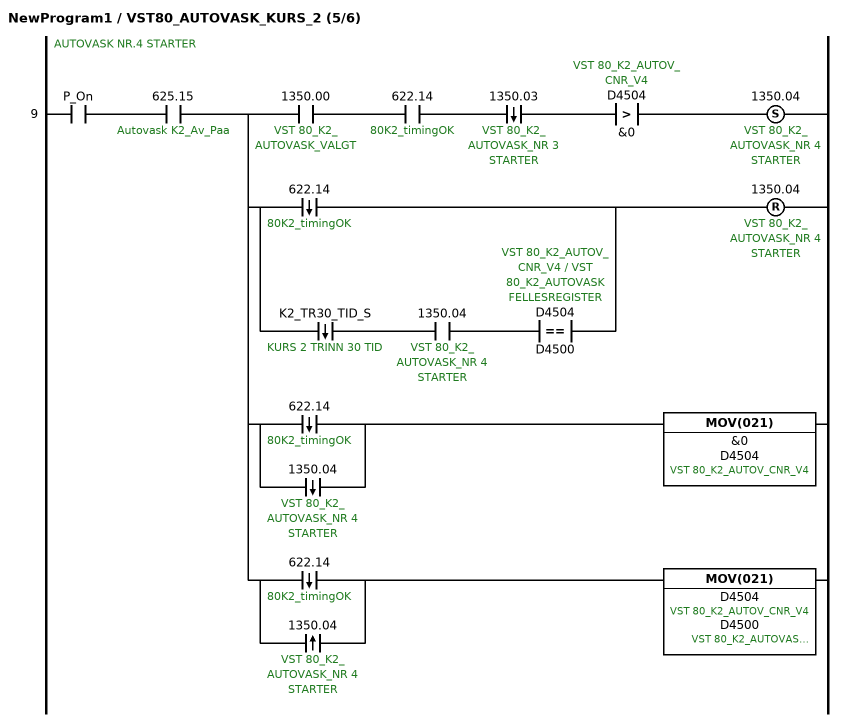
; [picture p288: NewProgram1 / VST80_AUTOVASK_KURS_2, rungs 9-9]
; rung 9: AUTOVASK NR.4 STARTER
LD P_On
AND 625.15  ; Autovask K2_Av_Paa
OUT TR0
AND 1350.00  ; VST 80_K2_AUTOVASK_VALGT
AND 622.14  ; 80K2_timingOK
%AND 1350.03  ; VST 80_K2_AUTOVASK_NR 3 STARTER
AND>(320) D4504 &0  ; VST 80_K2_AUTOV_CNR_V4
SET 1350.04  ; VST 80_K2_AUTOVASK_NR 4 STARTER
LD TR0
%LD 622.14  ; 80K2_timingOK
%LD K2_TR30_TID_S  ; KURS 2 TRINN 30 TID
AND 1350.04  ; VST 80_K2_AUTOVASK_NR 4 STARTER
AND=(300) D4504 D4500  ; VST 80_K2_AUTOV_CNR_V4, VST 80_K2_AUTOVASK FELLESREGISTER
ORLD
ANDLD
RSET 1350.04  ; VST 80_K2_AUTOVASK_NR 4 STARTER
LD TR0
%LD 622.14  ; 80K2_timingOK
%OR 1350.04  ; VST 80_K2_AUTOVASK_NR 4 STARTER
ANDLD
MOV(021) &0 D4504  ; VST 80_K2_AUTOV_CNR_V4
LD TR0
%LD 622.14  ; 80K2_timingOK
@OR 1350.04  ; VST 80_K2_AUTOVASK_NR 4 STARTER
ANDLD
MOV(021) D4504 D4500  ; VST 80_K2_AUTOV_CNR_V4, VST 80_K2_AUTOVASK FELLESREGISTER

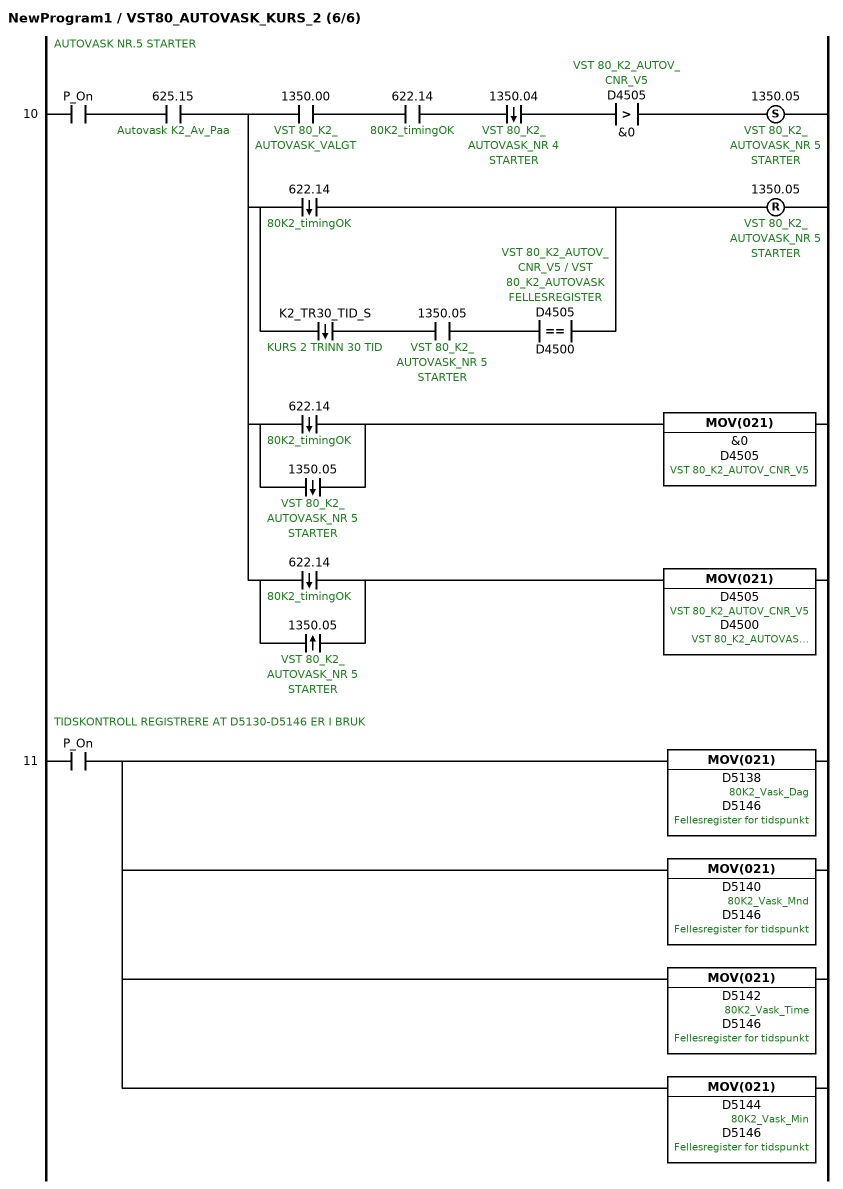
; rung 10: AUTOVASK NR.5 STARTER
LD P_On
AND 625.15  ; Autovask K2_Av_Paa
OUT TR0
AND 1350.00  ; VST 80_K2_AUTOVASK_VALGT
AND 622.14  ; 80K2_timingOK
%AND 1350.04  ; VST 80_K2_AUTOVASK_NR 4 STARTER
AND>(320) D4505 &0  ; VST 80_K2_AUTOV_CNR_V5
SET 1350.05  ; VST 80_K2_AUTOVASK_NR 5 STARTER
LD TR0
%LD 622.14  ; 80K2_timingOK
%LD K2_TR30_TID_S  ; KURS 2 TRINN 30 TID
AND 1350.05  ; VST 80_K2_AUTOVASK_NR 5 STARTER
AND=(300) D4505 D4500  ; VST 80_K2_AUTOV_CNR_V5, VST 80_K2_AUTOVASK FELLESREGISTER
ORLD
ANDLD
RSET 1350.05  ; VST 80_K2_AUTOVASK_NR 5 STARTER
LD TR0
%LD 622.14  ; 80K2_timingOK
%OR 1350.05  ; VST 80_K2_AUTOVASK_NR 5 STARTER
ANDLD
MOV(021) &0 D4505  ; VST 80_K2_AUTOV_CNR_V5
LD TR0
%LD 622.14  ; 80K2_timingOK
@OR 1350.05  ; VST 80_K2_AUTOVASK_NR 5 STARTER
ANDLD
MOV(021) D4505 D4500  ; VST 80_K2_AUTOV_CNR_V5, VST 80_K2_AUTOVASK FELLESREGISTER
; rung 11: TIDSKONTROLL REGISTRERE AT D5130-D5146 ER I BRUK
LD P_On
MOV(021) D5138 D5146  ; 80K2_Vask_Dag, Fellesregister for tidspunkt
MOV(021) D5140 D5146  ; 80K2_Vask_Mnd, Fellesregister for tidspunkt
MOV(021) D5142 D5146  ; 80K2_Vask_Time, Fellesregister for tidspunkt
MOV(021) D5144 D5146  ; 80K2_Vask_Min, Fellesregister for tidspunkt
; rung 12: Ingen_kommentar_funnet

### Section VST80_K_3_TIDER_TR1_18

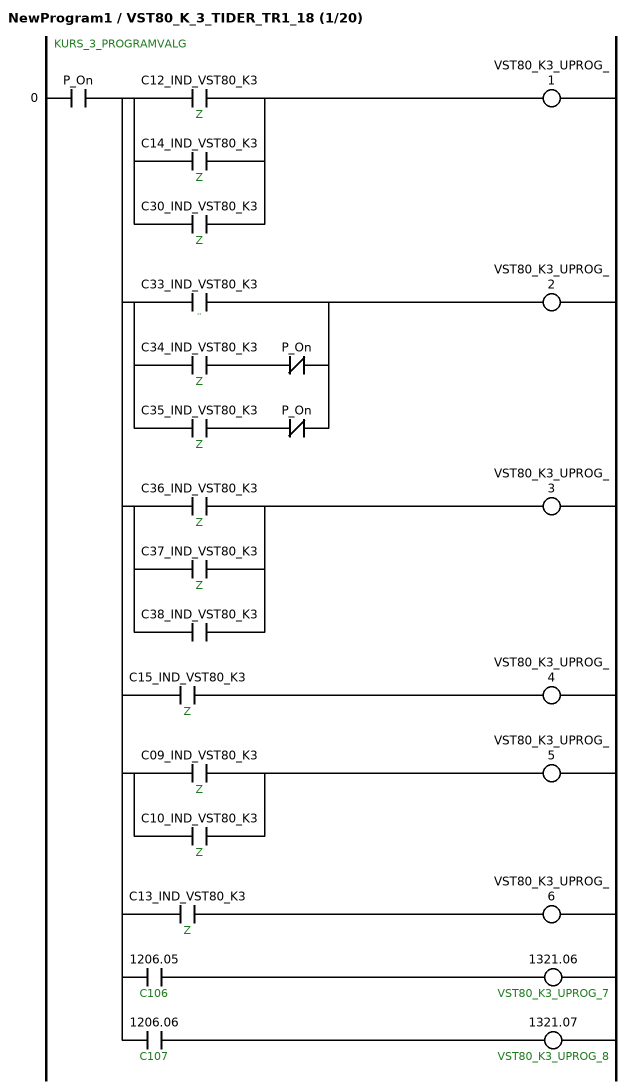
; rung 0: KURS_3_PROGRAMVALG
LD P_On
OUT TR0
LD C12_IND_VST80_K3  ; Z
OR C14_IND_VST80_K3  ; Z
OR C30_IND_VST80_K3  ; Z
ANDLD
OUT VST80_K3_UPROG_1
LD TR0
LD C33_IND_VST80_K3  ; ¨
LD C34_IND_VST80_K3  ; Z
ANDNOT P_On
ORLD
LD C35_IND_VST80_K3  ; Z
ANDNOT P_On
ORLD
ANDLD
OUT VST80_K3_UPROG_2
LD TR0
LD C36_IND_VST80_K3  ; Z
OR C37_IND_VST80_K3  ; Z
OR C38_IND_VST80_K3
ANDLD
OUT VST80_K3_UPROG_3
LD TR0
AND C15_IND_VST80_K3  ; Z
OUT VST80_K3_UPROG_4
LD TR0
LD C09_IND_VST80_K3  ; Z
OR C10_IND_VST80_K3  ; Z
ANDLD
OUT VST80_K3_UPROG_5
LD TR0
AND C13_IND_VST80_K3  ; Z
OUT VST80_K3_UPROG_6
LD TR0
AND 1206.05  ; C106
OUT 1321.06  ; VST80_K3_UPROG_7
LD TR0
AND 1206.06  ; C107
OUT 1321.07  ; VST80_K3_UPROG_8

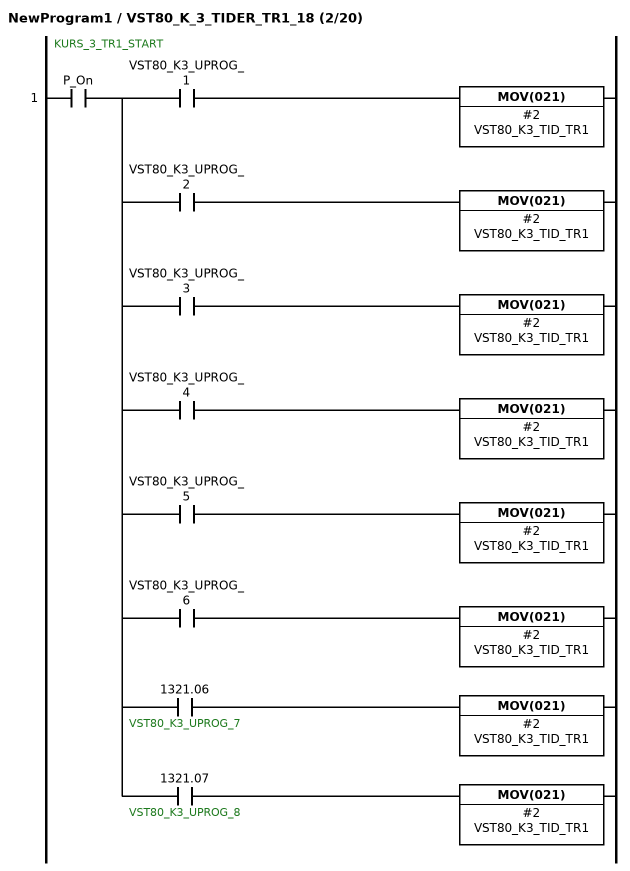
; rung 1: KURS_3_TR1_START
LD P_On
OUT TR0
AND VST80_K3_UPROG_1
MOV(021) #2 VST80_K3_TID_TR1
LD TR0
AND VST80_K3_UPROG_2
MOV(021) #2 VST80_K3_TID_TR1
LD TR0
AND VST80_K3_UPROG_3
MOV(021) #2 VST80_K3_TID_TR1
LD TR0
AND VST80_K3_UPROG_4
MOV(021) #2 VST80_K3_TID_TR1
LD TR0
AND VST80_K3_UPROG_5
MOV(021) #2 VST80_K3_TID_TR1
LD TR0
AND VST80_K3_UPROG_6
MOV(021) #2 VST80_K3_TID_TR1
LD TR0
AND 1321.06  ; VST80_K3_UPROG_7
MOV(021) #2 VST80_K3_TID_TR1
LD TR0
AND 1321.07  ; VST80_K3_UPROG_8
MOV(021) #2 VST80_K3_TID_TR1

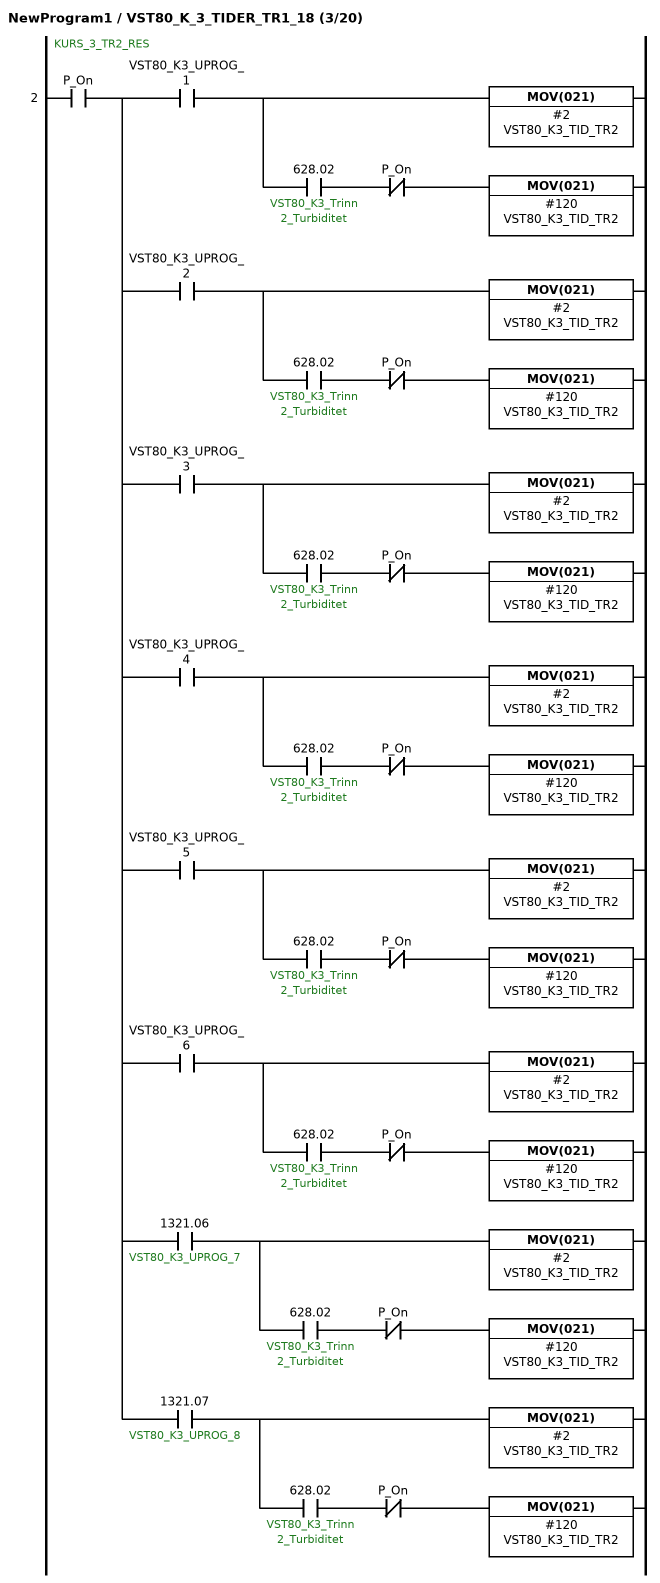
; rung 2: KURS_3_TR2_RES
LD P_On
OUT TR0
AND VST80_K3_UPROG_1
MOV(021) #2 VST80_K3_TID_TR2
AND 628.02  ; VST80_K3_Trinn 2_Turbiditet
ANDNOT P_On
MOV(021) #120 VST80_K3_TID_TR2
LD TR0
AND VST80_K3_UPROG_2
MOV(021) #2 VST80_K3_TID_TR2
AND 628.02  ; VST80_K3_Trinn 2_Turbiditet
ANDNOT P_On
MOV(021) #120 VST80_K3_TID_TR2
LD TR0
AND VST80_K3_UPROG_3
MOV(021) #2 VST80_K3_TID_TR2
AND 628.02  ; VST80_K3_Trinn 2_Turbiditet
ANDNOT P_On
MOV(021) #120 VST80_K3_TID_TR2
LD TR0
AND VST80_K3_UPROG_4
MOV(021) #2 VST80_K3_TID_TR2
AND 628.02  ; VST80_K3_Trinn 2_Turbiditet
ANDNOT P_On
MOV(021) #120 VST80_K3_TID_TR2
LD TR0
AND VST80_K3_UPROG_5
MOV(021) #2 VST80_K3_TID_TR2
AND 628.02  ; VST80_K3_Trinn 2_Turbiditet
ANDNOT P_On
MOV(021) #120 VST80_K3_TID_TR2
LD TR0
AND VST80_K3_UPROG_6
MOV(021) #2 VST80_K3_TID_TR2
AND 628.02  ; VST80_K3_Trinn 2_Turbiditet
ANDNOT P_On
MOV(021) #120 VST80_K3_TID_TR2
LD TR0
AND 1321.06  ; VST80_K3_UPROG_7
MOV(021) #2 VST80_K3_TID_TR2
AND 628.02  ; VST80_K3_Trinn 2_Turbiditet
ANDNOT P_On
MOV(021) #120 VST80_K3_TID_TR2
LD TR0
AND 1321.07  ; VST80_K3_UPROG_8
MOV(021) #2 VST80_K3_TID_TR2
AND 628.02  ; VST80_K3_Trinn 2_Turbiditet
ANDNOT P_On
MOV(021) #120 VST80_K3_TID_TR2

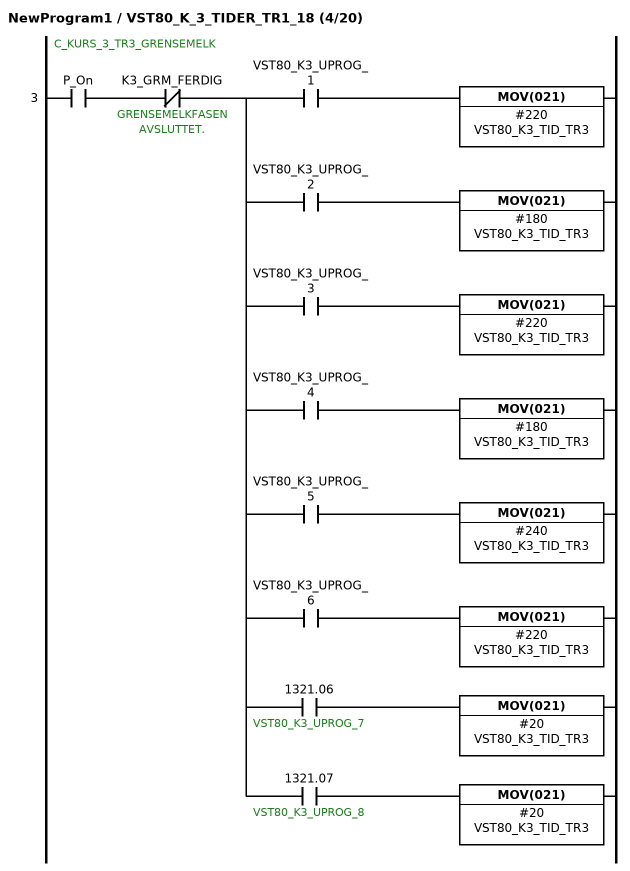
; rung 3: C_KURS_3_TR3_GRENSEMELK
LD P_On
ANDNOT K3_GRM_FERDIG  ; GRENSEMELKFASEN AVSLUTTET.
OUT TR0
AND VST80_K3_UPROG_1
MOV(021) #220 VST80_K3_TID_TR3
LD TR0
AND VST80_K3_UPROG_2
MOV(021) #180 VST80_K3_TID_TR3
LD TR0
AND VST80_K3_UPROG_3
MOV(021) #220 VST80_K3_TID_TR3
LD TR0
AND VST80_K3_UPROG_4
MOV(021) #180 VST80_K3_TID_TR3
LD TR0
AND VST80_K3_UPROG_5
MOV(021) #240 VST80_K3_TID_TR3
LD TR0
AND VST80_K3_UPROG_6
MOV(021) #220 VST80_K3_TID_TR3
LD TR0
AND 1321.06  ; VST80_K3_UPROG_7
MOV(021) #20 VST80_K3_TID_TR3
LD TR0
AND 1321.07  ; VST80_K3_UPROG_8
MOV(021) #20 VST80_K3_TID_TR3

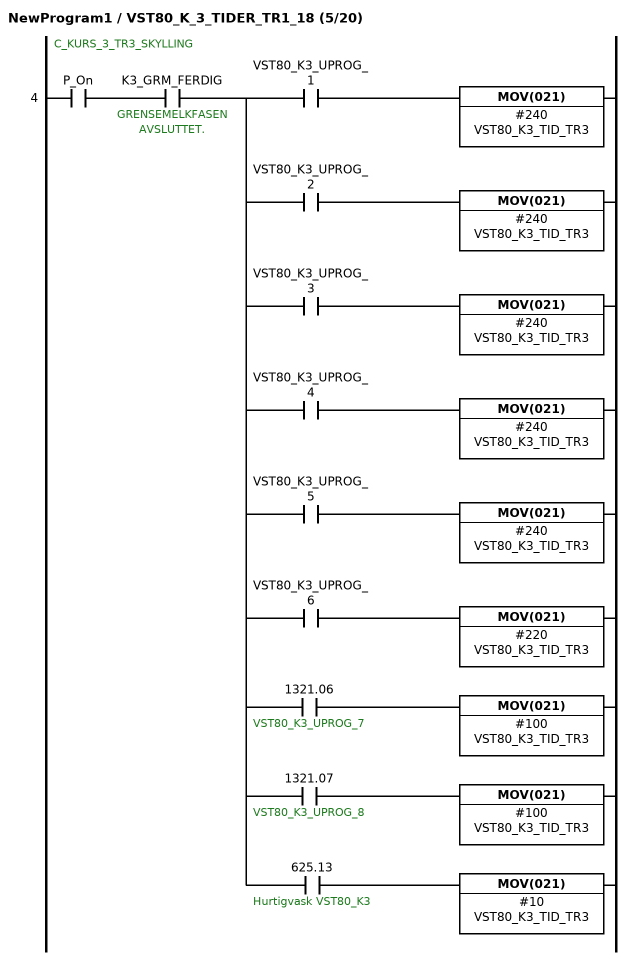
; rung 4: C_KURS_3_TR3_SKYLLING
LD P_On
AND K3_GRM_FERDIG  ; GRENSEMELKFASEN AVSLUTTET.
OUT TR0
AND VST80_K3_UPROG_1
MOV(021) #240 VST80_K3_TID_TR3
LD TR0
AND VST80_K3_UPROG_2
MOV(021) #240 VST80_K3_TID_TR3
LD TR0
AND VST80_K3_UPROG_3
MOV(021) #240 VST80_K3_TID_TR3
LD TR0
AND VST80_K3_UPROG_4
MOV(021) #240 VST80_K3_TID_TR3
LD TR0
AND VST80_K3_UPROG_5
MOV(021) #240 VST80_K3_TID_TR3
LD TR0
AND VST80_K3_UPROG_6
MOV(021) #220 VST80_K3_TID_TR3
LD TR0
AND 1321.06  ; VST80_K3_UPROG_7
MOV(021) #100 VST80_K3_TID_TR3
LD TR0
AND 1321.07  ; VST80_K3_UPROG_8
MOV(021) #100 VST80_K3_TID_TR3
LD TR0
AND 625.13  ; Hurtigvask VST80_K3
MOV(021) #10 VST80_K3_TID_TR3

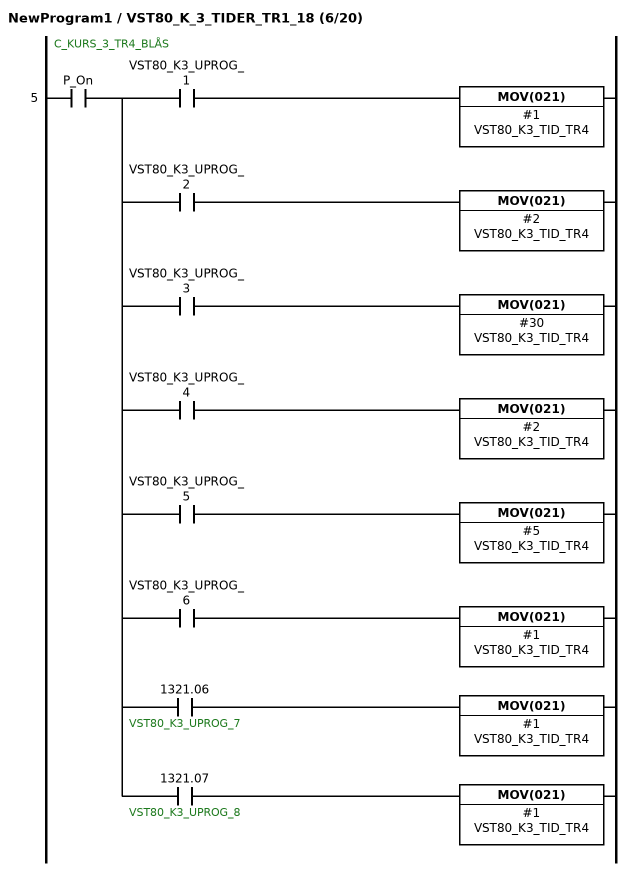
; rung 5: C_KURS_3_TR4_BLÅS
LD P_On
OUT TR0
AND VST80_K3_UPROG_1
MOV(021) #1 VST80_K3_TID_TR4
LD TR0
AND VST80_K3_UPROG_2
MOV(021) #2 VST80_K3_TID_TR4
LD TR0
AND VST80_K3_UPROG_3
MOV(021) #30 VST80_K3_TID_TR4
LD TR0
AND VST80_K3_UPROG_4
MOV(021) #2 VST80_K3_TID_TR4
LD TR0
AND VST80_K3_UPROG_5
MOV(021) #5 VST80_K3_TID_TR4
LD TR0
AND VST80_K3_UPROG_6
MOV(021) #1 VST80_K3_TID_TR4
LD TR0
AND 1321.06  ; VST80_K3_UPROG_7
MOV(021) #1 VST80_K3_TID_TR4
LD TR0
AND 1321.07  ; VST80_K3_UPROG_8
MOV(021) #1 VST80_K3_TID_TR4

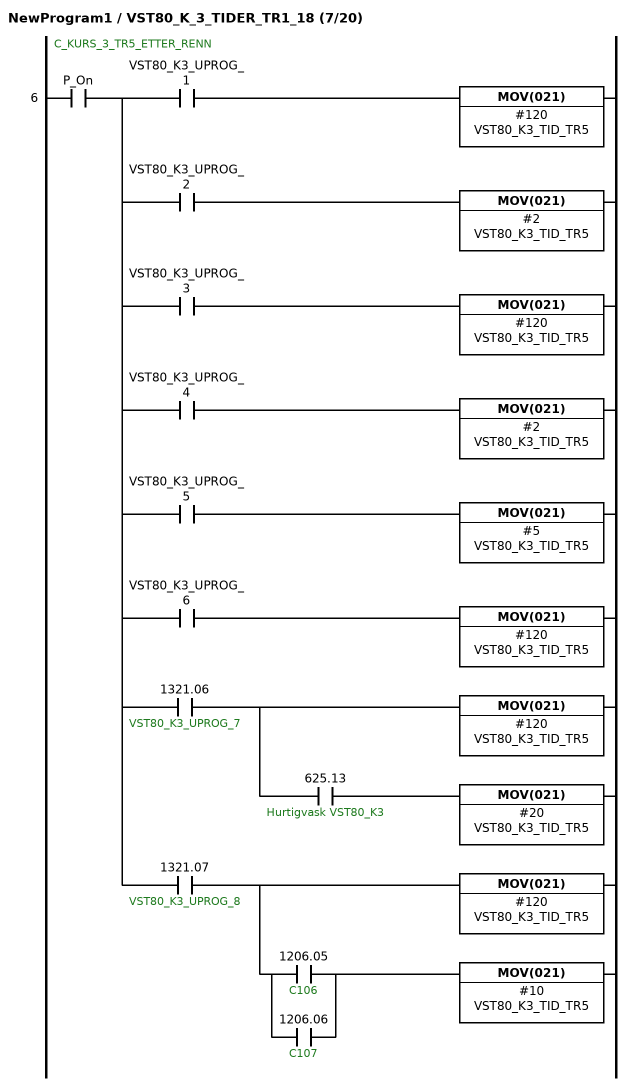
; rung 6: C_KURS_3_TR5_ETTER_RENN
LD P_On
OUT TR0
AND VST80_K3_UPROG_1
MOV(021) #120 VST80_K3_TID_TR5
LD TR0
AND VST80_K3_UPROG_2
MOV(021) #2 VST80_K3_TID_TR5
LD TR0
AND VST80_K3_UPROG_3
MOV(021) #120 VST80_K3_TID_TR5
LD TR0
AND VST80_K3_UPROG_4
MOV(021) #2 VST80_K3_TID_TR5
LD TR0
AND VST80_K3_UPROG_5
MOV(021) #5 VST80_K3_TID_TR5
LD TR0
AND VST80_K3_UPROG_6
MOV(021) #120 VST80_K3_TID_TR5
LD TR0
AND 1321.06  ; VST80_K3_UPROG_7
MOV(021) #120 VST80_K3_TID_TR5
AND 625.13  ; Hurtigvask VST80_K3
MOV(021) #20 VST80_K3_TID_TR5
LD TR0
AND 1321.07  ; VST80_K3_UPROG_8
MOV(021) #120 VST80_K3_TID_TR5
LD 1206.05  ; C106
OR 1206.06  ; C107
ANDLD
MOV(021) #10 VST80_K3_TID_TR5

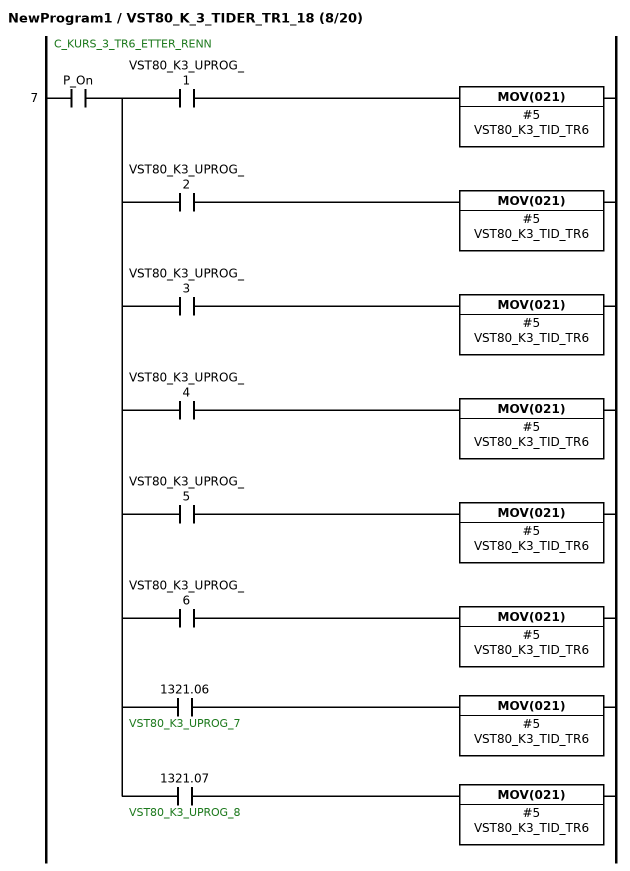
; rung 7: C_KURS_3_TR6_ETTER_RENN
LD P_On
OUT TR0
AND VST80_K3_UPROG_1
MOV(021) #5 VST80_K3_TID_TR6
LD TR0
AND VST80_K3_UPROG_2
MOV(021) #5 VST80_K3_TID_TR6
LD TR0
AND VST80_K3_UPROG_3
MOV(021) #5 VST80_K3_TID_TR6
LD TR0
AND VST80_K3_UPROG_4
MOV(021) #5 VST80_K3_TID_TR6
LD TR0
AND VST80_K3_UPROG_5
MOV(021) #5 VST80_K3_TID_TR6
LD TR0
AND VST80_K3_UPROG_6
MOV(021) #5 VST80_K3_TID_TR6
LD TR0
AND 1321.06  ; VST80_K3_UPROG_7
MOV(021) #5 VST80_K3_TID_TR6
LD TR0
AND 1321.07  ; VST80_K3_UPROG_8
MOV(021) #5 VST80_K3_TID_TR6

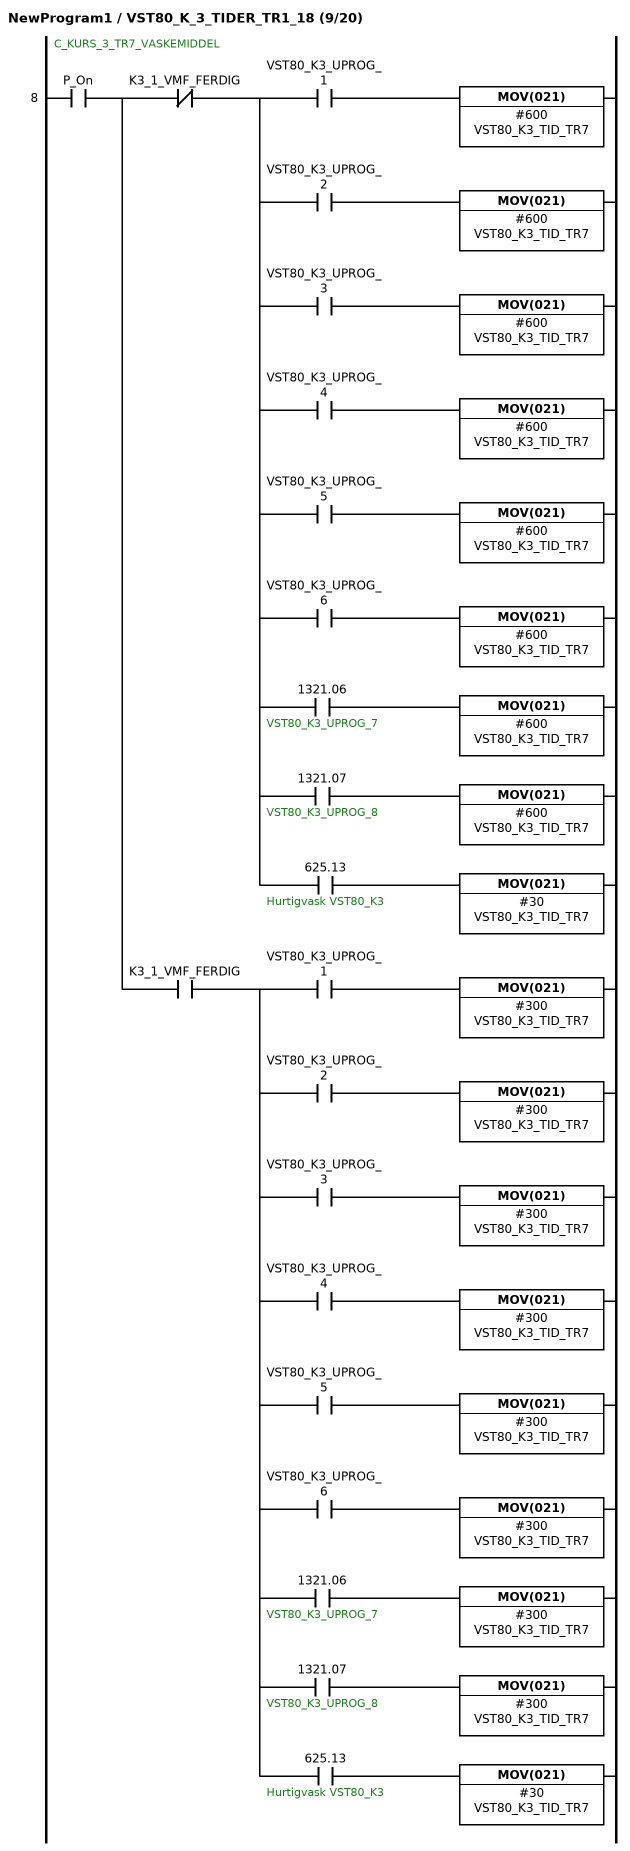
; rung 8: C_KURS_3_TR7_VASKEMIDDEL
LD P_On
OUT TR0
ANDNOT K3_1_VMF_FERDIG
OUT TR1
AND VST80_K3_UPROG_1
MOV(021) #600 VST80_K3_TID_TR7
LD TR1
AND VST80_K3_UPROG_2
MOV(021) #600 VST80_K3_TID_TR7
LD TR1
AND VST80_K3_UPROG_3
MOV(021) #600 VST80_K3_TID_TR7
LD TR1
AND VST80_K3_UPROG_4
MOV(021) #600 VST80_K3_TID_TR7
LD TR1
AND VST80_K3_UPROG_5
MOV(021) #600 VST80_K3_TID_TR7
LD TR1
AND VST80_K3_UPROG_6
MOV(021) #600 VST80_K3_TID_TR7
LD TR1
AND 1321.06  ; VST80_K3_UPROG_7
MOV(021) #600 VST80_K3_TID_TR7
LD TR1
AND 1321.07  ; VST80_K3_UPROG_8
MOV(021) #600 VST80_K3_TID_TR7
LD TR1
AND 625.13  ; Hurtigvask VST80_K3
MOV(021) #30 VST80_K3_TID_TR7
LD TR0
AND K3_1_VMF_FERDIG
OUT TR0
AND VST80_K3_UPROG_1
MOV(021) #300 VST80_K3_TID_TR7
LD TR0
AND VST80_K3_UPROG_2
MOV(021) #300 VST80_K3_TID_TR7
LD TR0
AND VST80_K3_UPROG_3
MOV(021) #300 VST80_K3_TID_TR7
LD TR0
AND VST80_K3_UPROG_4
MOV(021) #300 VST80_K3_TID_TR7
LD TR0
AND VST80_K3_UPROG_5
MOV(021) #300 VST80_K3_TID_TR7
LD TR0
AND VST80_K3_UPROG_6
MOV(021) #300 VST80_K3_TID_TR7
LD TR0
AND 1321.06  ; VST80_K3_UPROG_7
MOV(021) #300 VST80_K3_TID_TR7
LD TR0
AND 1321.07  ; VST80_K3_UPROG_8
MOV(021) #300 VST80_K3_TID_TR7
LD TR0
AND 625.13  ; Hurtigvask VST80_K3
MOV(021) #30 VST80_K3_TID_TR7

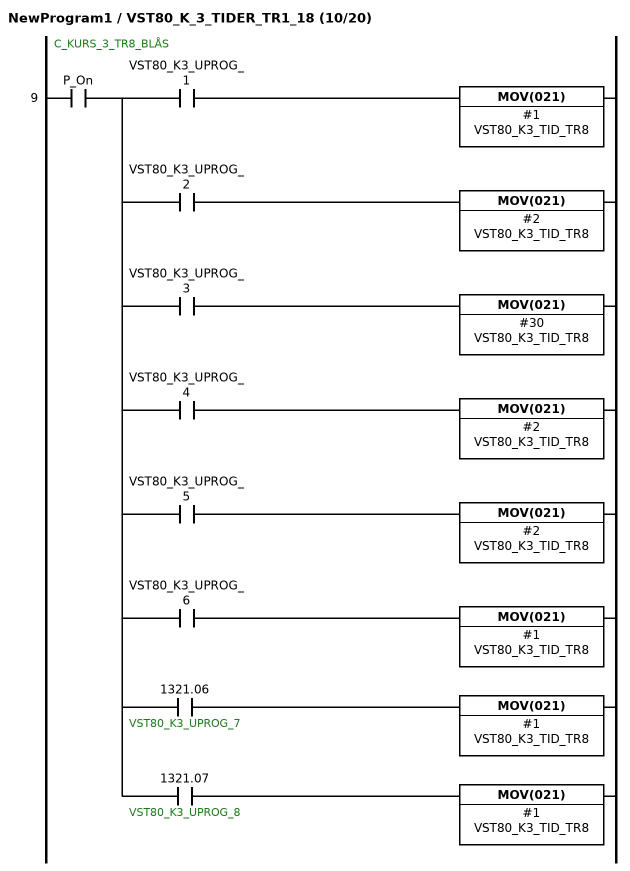
; rung 9: C_KURS_3_TR8_BLÅS
LD P_On
OUT TR0
AND VST80_K3_UPROG_1
MOV(021) #1 VST80_K3_TID_TR8
LD TR0
AND VST80_K3_UPROG_2
MOV(021) #2 VST80_K3_TID_TR8
LD TR0
AND VST80_K3_UPROG_3
MOV(021) #30 VST80_K3_TID_TR8
LD TR0
AND VST80_K3_UPROG_4
MOV(021) #2 VST80_K3_TID_TR8
LD TR0
AND VST80_K3_UPROG_5
MOV(021) #2 VST80_K3_TID_TR8
LD TR0
AND VST80_K3_UPROG_6
MOV(021) #1 VST80_K3_TID_TR8
LD TR0
AND 1321.06  ; VST80_K3_UPROG_7
MOV(021) #1 VST80_K3_TID_TR8
LD TR0
AND 1321.07  ; VST80_K3_UPROG_8
MOV(021) #1 VST80_K3_TID_TR8

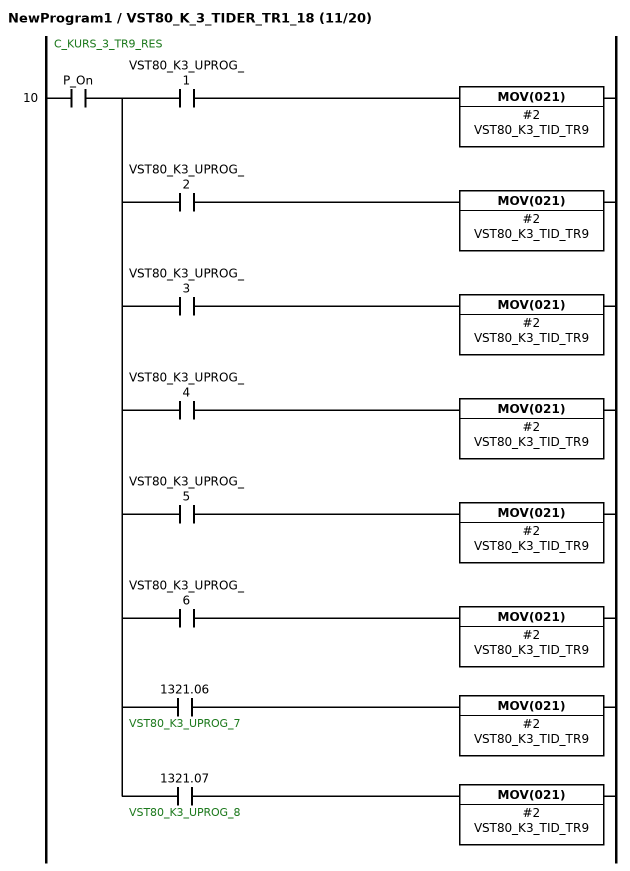
; rung 10: C_KURS_3_TR9_RES
LD P_On
OUT TR0
AND VST80_K3_UPROG_1
MOV(021) #2 VST80_K3_TID_TR9
LD TR0
AND VST80_K3_UPROG_2
MOV(021) #2 VST80_K3_TID_TR9
LD TR0
AND VST80_K3_UPROG_3
MOV(021) #2 VST80_K3_TID_TR9
LD TR0
AND VST80_K3_UPROG_4
MOV(021) #2 VST80_K3_TID_TR9
LD TR0
AND VST80_K3_UPROG_5
MOV(021) #2 VST80_K3_TID_TR9
LD TR0
AND VST80_K3_UPROG_6
MOV(021) #2 VST80_K3_TID_TR9
LD TR0
AND 1321.06  ; VST80_K3_UPROG_7
MOV(021) #2 VST80_K3_TID_TR9
LD TR0
AND 1321.07  ; VST80_K3_UPROG_8
MOV(021) #2 VST80_K3_TID_TR9

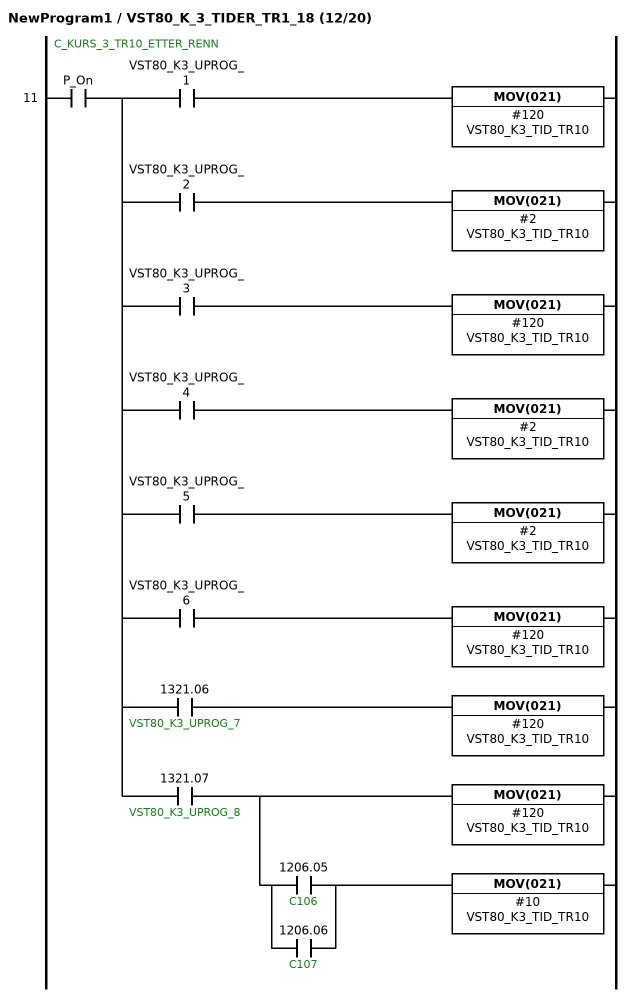
; rung 11: C_KURS_3_TR10_ETTER_RENN
LD P_On
OUT TR0
AND VST80_K3_UPROG_1
MOV(021) #120 VST80_K3_TID_TR10
LD TR0
AND VST80_K3_UPROG_2
MOV(021) #2 VST80_K3_TID_TR10
LD TR0
AND VST80_K3_UPROG_3
MOV(021) #120 VST80_K3_TID_TR10
LD TR0
AND VST80_K3_UPROG_4
MOV(021) #2 VST80_K3_TID_TR10
LD TR0
AND VST80_K3_UPROG_5
MOV(021) #2 VST80_K3_TID_TR10
LD TR0
AND VST80_K3_UPROG_6
MOV(021) #120 VST80_K3_TID_TR10
LD TR0
AND 1321.06  ; VST80_K3_UPROG_7
MOV(021) #120 VST80_K3_TID_TR10
LD TR0
AND 1321.07  ; VST80_K3_UPROG_8
MOV(021) #120 VST80_K3_TID_TR10
LD 1206.05  ; C106
OR 1206.06  ; C107
ANDLD
MOV(021) #10 VST80_K3_TID_TR10

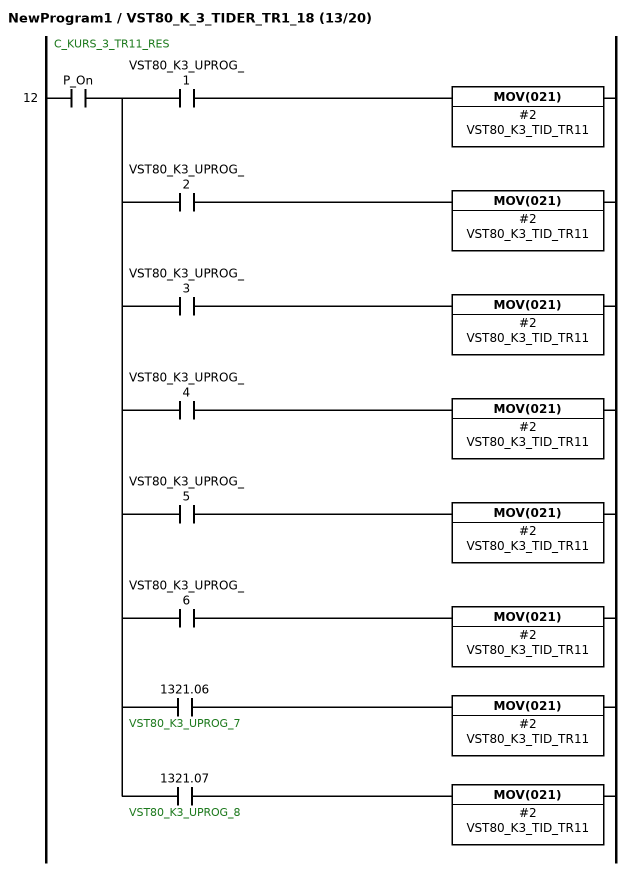
; rung 12: C_KURS_3_TR11_RES
LD P_On
OUT TR0
AND VST80_K3_UPROG_1
MOV(021) #2 VST80_K3_TID_TR11
LD TR0
AND VST80_K3_UPROG_2
MOV(021) #2 VST80_K3_TID_TR11
LD TR0
AND VST80_K3_UPROG_3
MOV(021) #2 VST80_K3_TID_TR11
LD TR0
AND VST80_K3_UPROG_4
MOV(021) #2 VST80_K3_TID_TR11
LD TR0
AND VST80_K3_UPROG_5
MOV(021) #2 VST80_K3_TID_TR11
LD TR0
AND VST80_K3_UPROG_6
MOV(021) #2 VST80_K3_TID_TR11
LD TR0
AND 1321.06  ; VST80_K3_UPROG_7
MOV(021) #2 VST80_K3_TID_TR11
LD TR0
AND 1321.07  ; VST80_K3_UPROG_8
MOV(021) #2 VST80_K3_TID_TR11

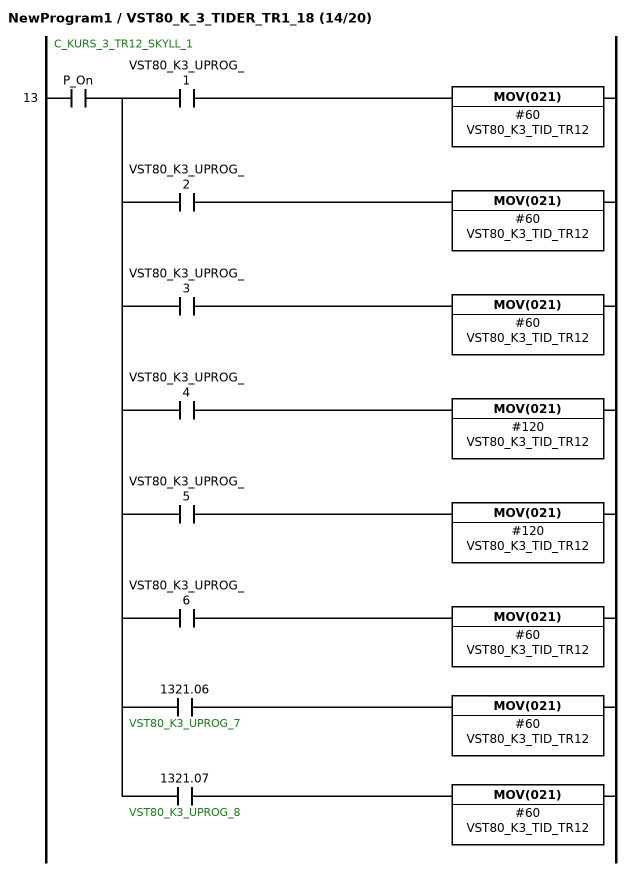
; rung 13: C_KURS_3_TR12_SKYLL_1
LD P_On
OUT TR0
AND VST80_K3_UPROG_1
MOV(021) #60 VST80_K3_TID_TR12
LD TR0
AND VST80_K3_UPROG_2
MOV(021) #60 VST80_K3_TID_TR12
LD TR0
AND VST80_K3_UPROG_3
MOV(021) #60 VST80_K3_TID_TR12
LD TR0
AND VST80_K3_UPROG_4
MOV(021) #120 VST80_K3_TID_TR12
LD TR0
AND VST80_K3_UPROG_5
MOV(021) #120 VST80_K3_TID_TR12
LD TR0
AND VST80_K3_UPROG_6
MOV(021) #60 VST80_K3_TID_TR12
LD TR0
AND 1321.06  ; VST80_K3_UPROG_7
MOV(021) #60 VST80_K3_TID_TR12
LD TR0
AND 1321.07  ; VST80_K3_UPROG_8
MOV(021) #60 VST80_K3_TID_TR12

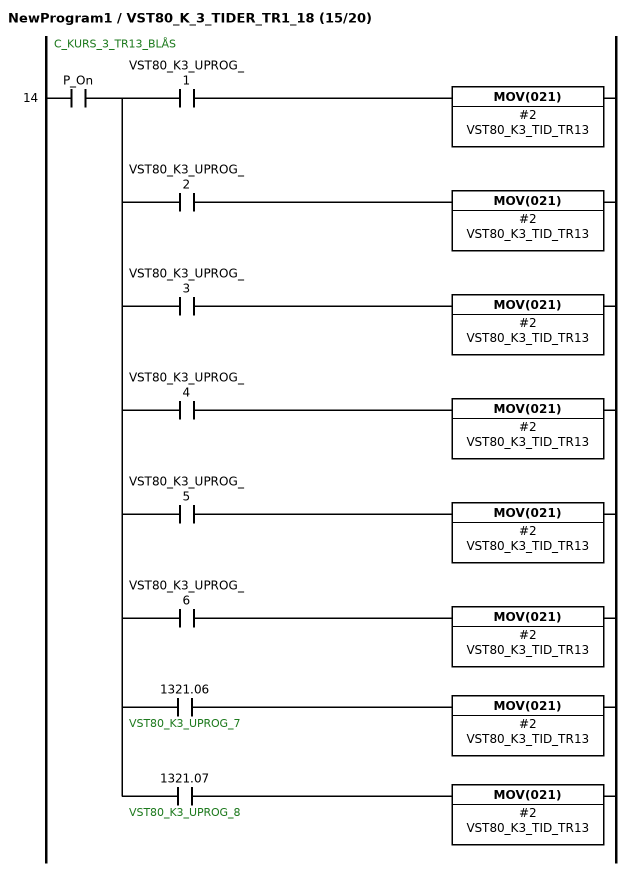
; rung 14: C_KURS_3_TR13_BLÅS
LD P_On
OUT TR0
AND VST80_K3_UPROG_1
MOV(021) #2 VST80_K3_TID_TR13
LD TR0
AND VST80_K3_UPROG_2
MOV(021) #2 VST80_K3_TID_TR13
LD TR0
AND VST80_K3_UPROG_3
MOV(021) #2 VST80_K3_TID_TR13
LD TR0
AND VST80_K3_UPROG_4
MOV(021) #2 VST80_K3_TID_TR13
LD TR0
AND VST80_K3_UPROG_5
MOV(021) #2 VST80_K3_TID_TR13
LD TR0
AND VST80_K3_UPROG_6
MOV(021) #2 VST80_K3_TID_TR13
LD TR0
AND 1321.06  ; VST80_K3_UPROG_7
MOV(021) #2 VST80_K3_TID_TR13
LD TR0
AND 1321.07  ; VST80_K3_UPROG_8
MOV(021) #2 VST80_K3_TID_TR13

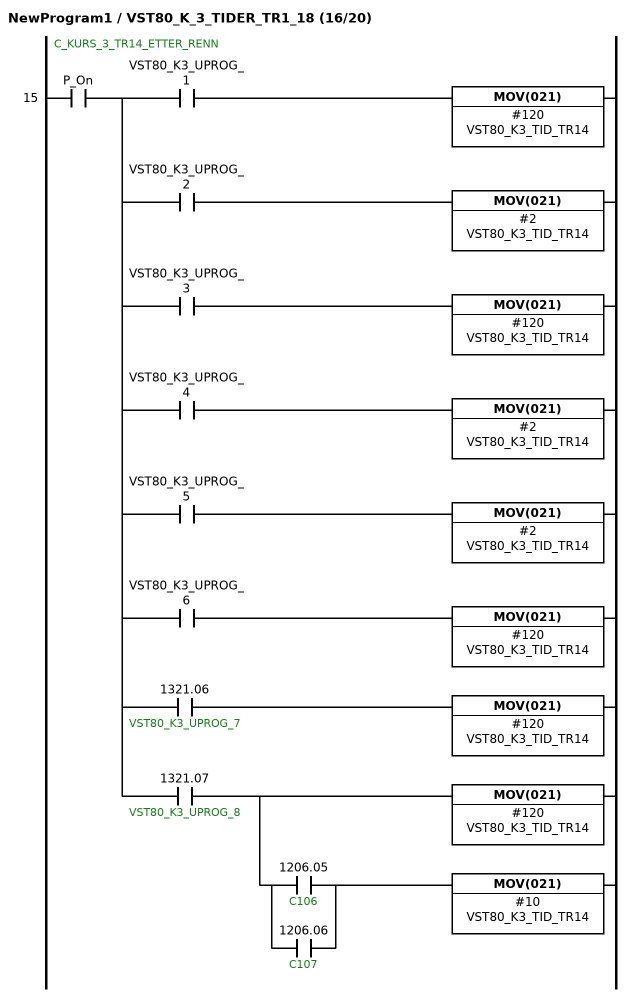
; rung 15: C_KURS_3_TR14_ETTER_RENN
LD P_On
OUT TR0
AND VST80_K3_UPROG_1
MOV(021) #120 VST80_K3_TID_TR14
LD TR0
AND VST80_K3_UPROG_2
MOV(021) #2 VST80_K3_TID_TR14
LD TR0
AND VST80_K3_UPROG_3
MOV(021) #120 VST80_K3_TID_TR14
LD TR0
AND VST80_K3_UPROG_4
MOV(021) #2 VST80_K3_TID_TR14
LD TR0
AND VST80_K3_UPROG_5
MOV(021) #2 VST80_K3_TID_TR14
LD TR0
AND VST80_K3_UPROG_6
MOV(021) #120 VST80_K3_TID_TR14
LD TR0
AND 1321.06  ; VST80_K3_UPROG_7
MOV(021) #120 VST80_K3_TID_TR14
LD TR0
AND 1321.07  ; VST80_K3_UPROG_8
MOV(021) #120 VST80_K3_TID_TR14
LD 1206.05  ; C106
OR 1206.06  ; C107
ANDLD
MOV(021) #10 VST80_K3_TID_TR14

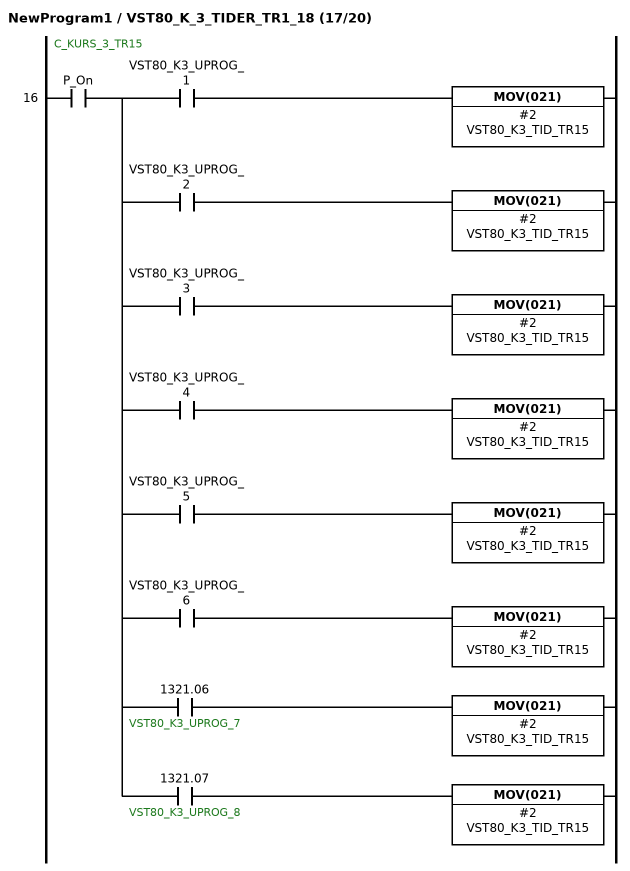
; rung 16: C_KURS_3_TR15
LD P_On
OUT TR0
AND VST80_K3_UPROG_1
MOV(021) #2 VST80_K3_TID_TR15
LD TR0
AND VST80_K3_UPROG_2
MOV(021) #2 VST80_K3_TID_TR15
LD TR0
AND VST80_K3_UPROG_3
MOV(021) #2 VST80_K3_TID_TR15
LD TR0
AND VST80_K3_UPROG_4
MOV(021) #2 VST80_K3_TID_TR15
LD TR0
AND VST80_K3_UPROG_5
MOV(021) #2 VST80_K3_TID_TR15
LD TR0
AND VST80_K3_UPROG_6
MOV(021) #2 VST80_K3_TID_TR15
LD TR0
AND 1321.06  ; VST80_K3_UPROG_7
MOV(021) #2 VST80_K3_TID_TR15
LD TR0
AND 1321.07  ; VST80_K3_UPROG_8
MOV(021) #2 VST80_K3_TID_TR15

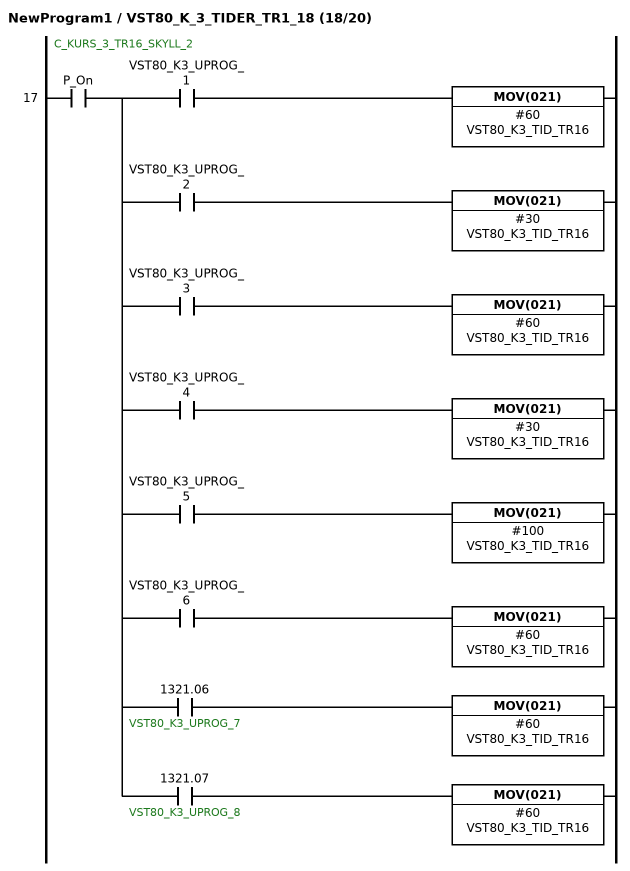
; rung 17: C_KURS_3_TR16_SKYLL_2
LD P_On
OUT TR0
AND VST80_K3_UPROG_1
MOV(021) #60 VST80_K3_TID_TR16
LD TR0
AND VST80_K3_UPROG_2
MOV(021) #30 VST80_K3_TID_TR16
LD TR0
AND VST80_K3_UPROG_3
MOV(021) #60 VST80_K3_TID_TR16
LD TR0
AND VST80_K3_UPROG_4
MOV(021) #30 VST80_K3_TID_TR16
LD TR0
AND VST80_K3_UPROG_5
MOV(021) #100 VST80_K3_TID_TR16
LD TR0
AND VST80_K3_UPROG_6
MOV(021) #60 VST80_K3_TID_TR16
LD TR0
AND 1321.06  ; VST80_K3_UPROG_7
MOV(021) #60 VST80_K3_TID_TR16
LD TR0
AND 1321.07  ; VST80_K3_UPROG_8
MOV(021) #60 VST80_K3_TID_TR16

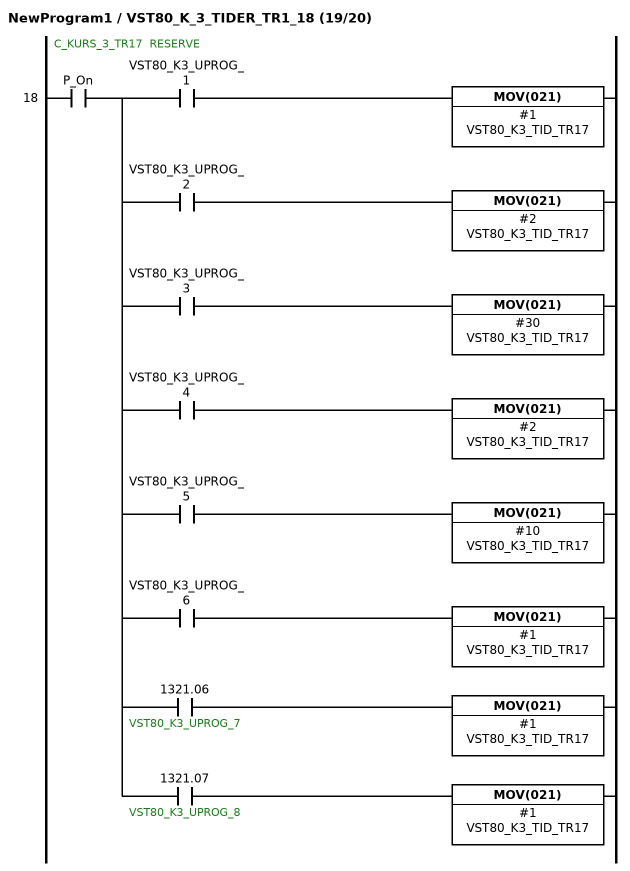
; rung 18: C_KURS_3_TR17  RESERVE
LD P_On
OUT TR0
AND VST80_K3_UPROG_1
MOV(021) #1 VST80_K3_TID_TR17
LD TR0
AND VST80_K3_UPROG_2
MOV(021) #2 VST80_K3_TID_TR17
LD TR0
AND VST80_K3_UPROG_3
MOV(021) #30 VST80_K3_TID_TR17
LD TR0
AND VST80_K3_UPROG_4
MOV(021) #2 VST80_K3_TID_TR17
LD TR0
AND VST80_K3_UPROG_5
MOV(021) #10 VST80_K3_TID_TR17
LD TR0
AND VST80_K3_UPROG_6
MOV(021) #1 VST80_K3_TID_TR17
LD TR0
AND 1321.06  ; VST80_K3_UPROG_7
MOV(021) #1 VST80_K3_TID_TR17
LD TR0
AND 1321.07  ; VST80_K3_UPROG_8
MOV(021) #1 VST80_K3_TID_TR17

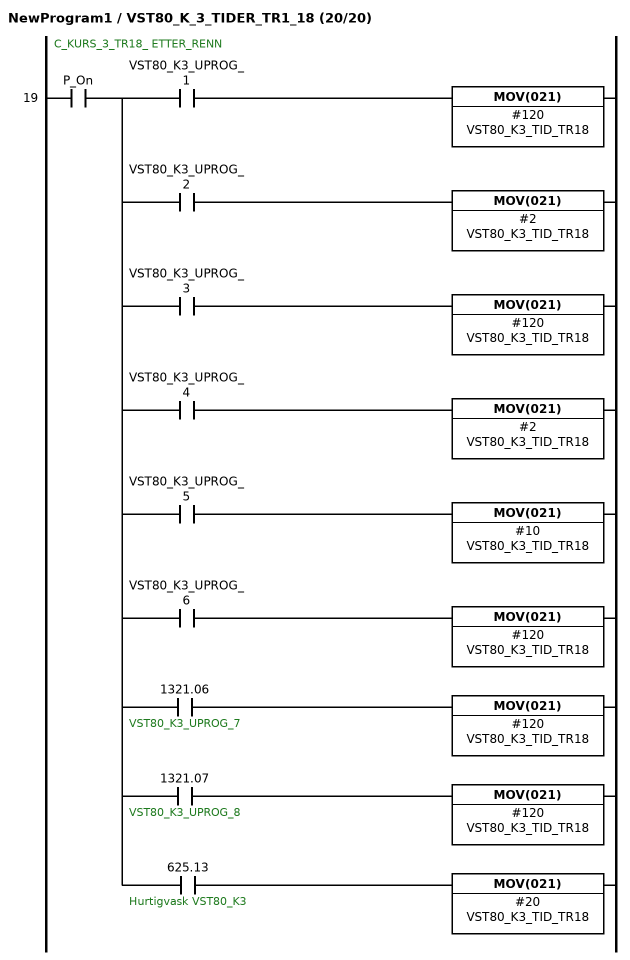
; rung 19: C_KURS_3_TR18_ ETTER_RENN
LD P_On
OUT TR0
AND VST80_K3_UPROG_1
MOV(021) #120 VST80_K3_TID_TR18
LD TR0
AND VST80_K3_UPROG_2
MOV(021) #2 VST80_K3_TID_TR18
LD TR0
AND VST80_K3_UPROG_3
MOV(021) #120 VST80_K3_TID_TR18
LD TR0
AND VST80_K3_UPROG_4
MOV(021) #2 VST80_K3_TID_TR18
LD TR0
AND VST80_K3_UPROG_5
MOV(021) #10 VST80_K3_TID_TR18
LD TR0
AND VST80_K3_UPROG_6
MOV(021) #120 VST80_K3_TID_TR18
LD TR0
AND 1321.06  ; VST80_K3_UPROG_7
MOV(021) #120 VST80_K3_TID_TR18
LD TR0
AND 1321.07  ; VST80_K3_UPROG_8
MOV(021) #120 VST80_K3_TID_TR18
LD TR0
AND 625.13  ; Hurtigvask VST80_K3
MOV(021) #20 VST80_K3_TID_TR18
; rung 20: Ingen_kommentar_funnet

### Section VST80_K_3_TIDER_TR19_30

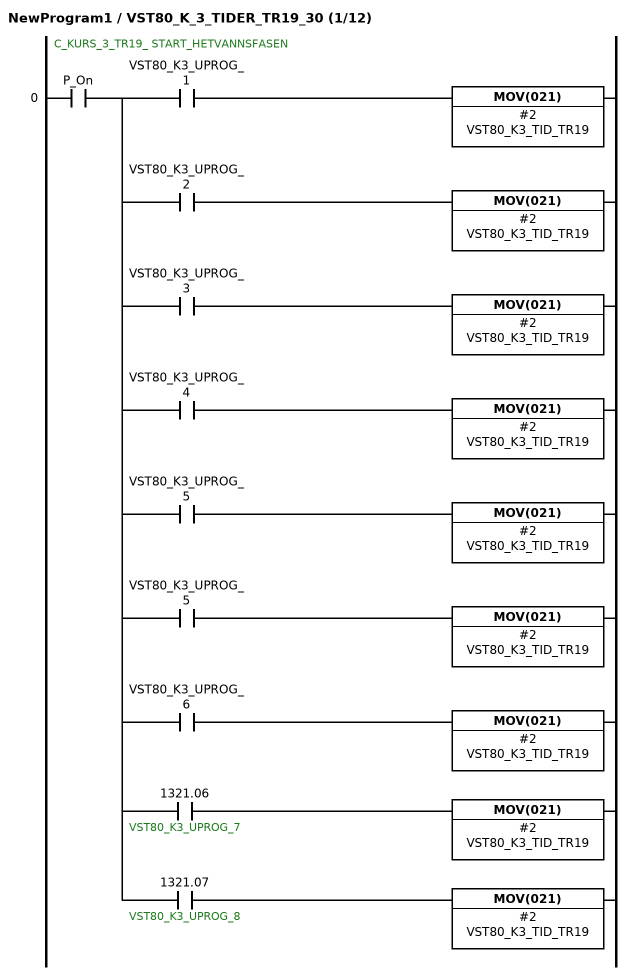
; rung 0: C_KURS_3_TR19_ START_HETVANNSFASEN
LD P_On
OUT TR0
AND VST80_K3_UPROG_1
MOV(021) #2 VST80_K3_TID_TR19
LD TR0
AND VST80_K3_UPROG_2
MOV(021) #2 VST80_K3_TID_TR19
LD TR0
AND VST80_K3_UPROG_3
MOV(021) #2 VST80_K3_TID_TR19
LD TR0
AND VST80_K3_UPROG_4
MOV(021) #2 VST80_K3_TID_TR19
LD TR0
AND VST80_K3_UPROG_5
MOV(021) #2 VST80_K3_TID_TR19
LD TR0
AND VST80_K3_UPROG_5
MOV(021) #2 VST80_K3_TID_TR19
LD TR0
AND VST80_K3_UPROG_6
MOV(021) #2 VST80_K3_TID_TR19
LD TR0
AND 1321.06  ; VST80_K3_UPROG_7
MOV(021) #2 VST80_K3_TID_TR19
LD TR0
AND 1321.07  ; VST80_K3_UPROG_8
MOV(021) #2 VST80_K3_TID_TR19

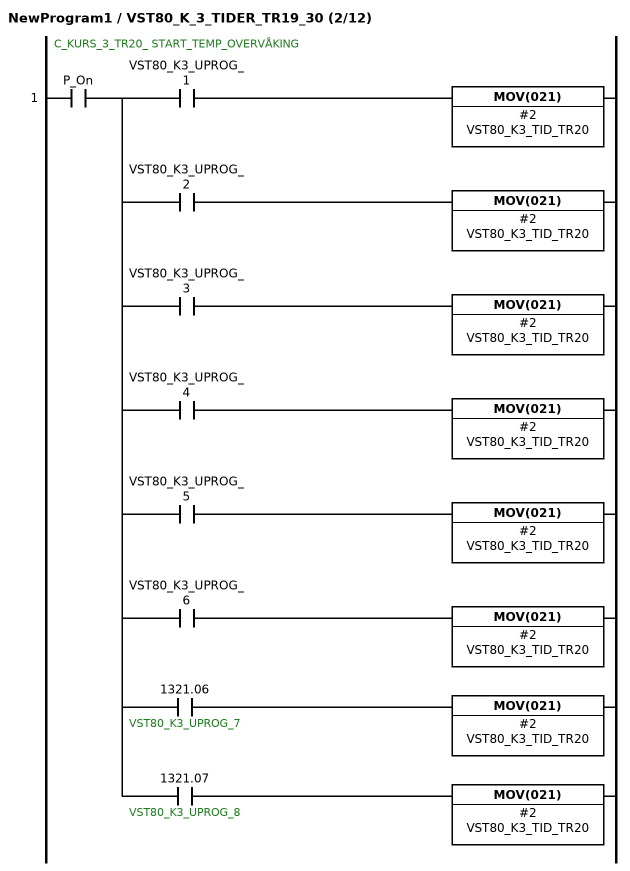
; rung 1: C_KURS_3_TR20_ START_TEMP_OVERVÅKING
LD P_On
OUT TR0
AND VST80_K3_UPROG_1
MOV(021) #2 VST80_K3_TID_TR20
LD TR0
AND VST80_K3_UPROG_2
MOV(021) #2 VST80_K3_TID_TR20
LD TR0
AND VST80_K3_UPROG_3
MOV(021) #2 VST80_K3_TID_TR20
LD TR0
AND VST80_K3_UPROG_4
MOV(021) #2 VST80_K3_TID_TR20
LD TR0
AND VST80_K3_UPROG_5
MOV(021) #2 VST80_K3_TID_TR20
LD TR0
AND VST80_K3_UPROG_6
MOV(021) #2 VST80_K3_TID_TR20
LD TR0
AND 1321.06  ; VST80_K3_UPROG_7
MOV(021) #2 VST80_K3_TID_TR20
LD TR0
AND 1321.07  ; VST80_K3_UPROG_8
MOV(021) #2 VST80_K3_TID_TR20

